//==================================================================================================
//							Beckhoff Automation Poland
//									18.05.2018
//	Struktura zawierajaca I/O odpowiedniego bloku
//  v1.0	|| TC v 3.1.4022.16		|| - pierwsza wersja
//==================================================================================================
TYPE ST_FBHoldingBrakeCtrlIO:
STRUCT
	bForceLock 						: BOOL;								// 
	bForceUnlock					: BOOL;								// 
	bBusy							: BOOL;
	bError							: BOOL; 							// General error: parameter or CoE read.
																		// If bError = TRUE and bInitialized = FALSE - error during read motor data.
																		// If bError = TRUE and bInitialized = TRUE and (iAdsErrId <> 0 or iCANopenErrId <> 0) then I2T read error
																		// If bError = TRUE and bInitialized = TRUE and iAdsErrId = 0 and iCANopenErrId = 0 then parameter error: rTorqueLimit outside permitted range rTorqueLimitLow..rTorqueLimitHigh or Empty stDriveRef
	uiAdsErrId						: UINT;								// Forwarded output FB_CoERead_ByDriveRef
	uiSecErrId						: UINT;								// Sercos Error ID for AX5000, CanOpen error ID for AX8000
END_STRUCT
END_TYPE

(* stored: Version 1.1.0.1, ProductVersion 3.1.4026.13, FileIdentifier 9c828baa3b1375ffcdf20bb480ad5787d400ea4e, FileSignature 4fc2dd48e08bb455d02eb5ee8721c2cbf7441a075081952cb086556decf487707db020af7755b88d8f694c992afd40d1de806a64b423aedb5068d293eb9e6f9711ea1ee21b218995673a2b9808f90caac7206026ca8e87f418dbeafed5d3085f1ea203f8da0281695a39c3cab7f92961c5ce2ee4047d91699f4605ecbe43fb149f83e07cc6b600a151e0233eed1fd5797da00c6699c49ea45c5cbdb7e1b08736f48ca57a4915ef956d41e4eb3d54821aae2fad72dc86841429c42f0de418aa653701ea64f1329e981f06f059b7e4d5fec8e0d4dd0162d250f3aa1dfea1e72bba0ff913eb9763673c882a3866046e5567d76bafb79d165cb2cba883e88c346a7a
   DUT ST_FBHoldingBrakeCtrlIO: Id {a71b2b00-1ef2-403e-b42a-9f3f34a37b0b} *)
